// TIA Portal project "Packaging of cubes" (V16)

(* hardware
DEVICE "HMI_1"  TP1200 Comfort
   slot 0: "HMI_1"  TP1200 Comfort  6AV2 124-0MC01-0AX0  16.0.0.0
   slot 1: "HMI_RT_1"  TP1200 Comfort  6AV2 124-0MC01-0AX0  16.0.0.0
   slot 5: "HMI_1.IE_CP_1"  PROFINET Interface  16.0.0.0
      slot 1: "PROFINET Interface_1"  PROFINET Interface
         slot 1: "Port_1"  Port
         slot 2: "Port_2"  Port
   slot 7: "HMI_1.MPI/DP_CP_1"  MPI/DP Interface  16.0.0.0
DEVICE "S71500/ET200MP station_1"  S7-1500 station
   slot 0: "Rail_0"  Rack  6ES7 590-1***0-0AA0
   slot 1: "PLC_1"  CPU 1511-1 PN  6ES7 511-1AK02-0AB0  V2.8
      slot 3: "CPU display_1"  6ES7591-1AA00-0AA0
      slot 32768: "PROFINET interface_1"  X1
         slot 32769: "Port_1"  X1 P1
         slot 32770: "Port_2"  X1 P2
      slot 34817: "Virtual CP interface port_1"  Virtual CP interface port  Virtual CP interface port
*)

// ===== PLC "PLC_1"  CPU 1511-1 PN =====

VAR_GLOBAL   // PLC tag table "Default tag table"
   "Green Cubes Sensor" AT %M0.0 : Bool;
   "Blue Cubes Sensor" AT %M0.1 : Bool;
   "Box not yet Full" AT %M0.2 : Bool;
   "Box Capacity" AT %M2.7 : Bool;
   "Upper Conveyor" AT %M0.4 : Bool;
   "Lower Conveyor" AT %M0.5 : Bool;
   "Box Conveyor" AT %M0.6 : Bool;
   "Box Changing" AT %M0.7 : Bool;
   "Start" AT %M2.0 : Bool;
   "PTRIG1" AT %M2.1 : Bool;
   "Box Sensor" AT %M2.2 : Bool;
   "PTRIG2" AT %M2.3 : Bool;
   "PTRIG3" AT %M2.4 : Bool;
   "PTRIG4" AT %M2.5 : Bool;
   "PTRIG5" AT %M2.6 : Bool;
   "toplam_kutu" AT %MW4 : Int;
   "ToplamMalzeme" AT %MW6 : Int;
   "PTRIG6" AT %M0.3 : Bool;
END_VAR

// folder: System blocks/Program resources

DATA_BLOCK "IEC_Counter_0_DB_2"   // DB1
{ S7_Optimized_Access := 'TRUE' }
AUTHOR : Simatic
FAMILY : IEC
NAME : CNTR
VERSION : 1.0
// stored: InstanceOfName IEC_COUNTER
"IEC_COUNTER"
BEGIN
END_DATA_BLOCK

DATA_BLOCK "IEC_Counter_0_DB"   // DB3
{ S7_Optimized_Access := 'TRUE' }
AUTHOR : Simatic
FAMILY : IEC
NAME : CNTR
VERSION : 1.0
// stored: InstanceOfName IEC_COUNTER
"IEC_COUNTER"
BEGIN
END_DATA_BLOCK

DATA_BLOCK "IEC_Counter_0_DB_1"   // DB4
{ S7_Optimized_Access := 'TRUE' }
AUTHOR : Simatic
FAMILY : IEC
NAME : CNTR
VERSION : 1.0
// stored: InstanceOfName IEC_COUNTER
"IEC_COUNTER"
BEGIN
END_DATA_BLOCK

DATA_BLOCK "IEC_Timer_0_DB_4"   // DB7
{ S7_Optimized_Access := 'TRUE' }
AUTHOR : Simatic
FAMILY : IEC
NAME : IEC_TMR
VERSION : 1.0
// stored: InstanceOfName IEC_TIMER
"IEC_TIMER"
BEGIN
END_DATA_BLOCK

// folder: (top level)

ORGANIZATION_BLOCK "Main"   // OB1, LAD, ProgramCycle
TITLE = "Main Program Sweep (Cycle)"
{ S7_Optimized_Access := 'TRUE' }
VERSION : 0.1
   VAR_INPUT
      Initial_Call : Bool;   // Initial call of this OB
      Remanence : Bool;   // =True, if remanent data are available
   END_VAR
   VAR_TEMP
      BoxCapacity1 : Bool;
   END_VAR
   VAR_TEMP   // added for the SCL form of the ladder/FBD networks
      _w1 : Bool;
      _w2 : Bool;
   END_VAR
BEGIN

REGION Network 1
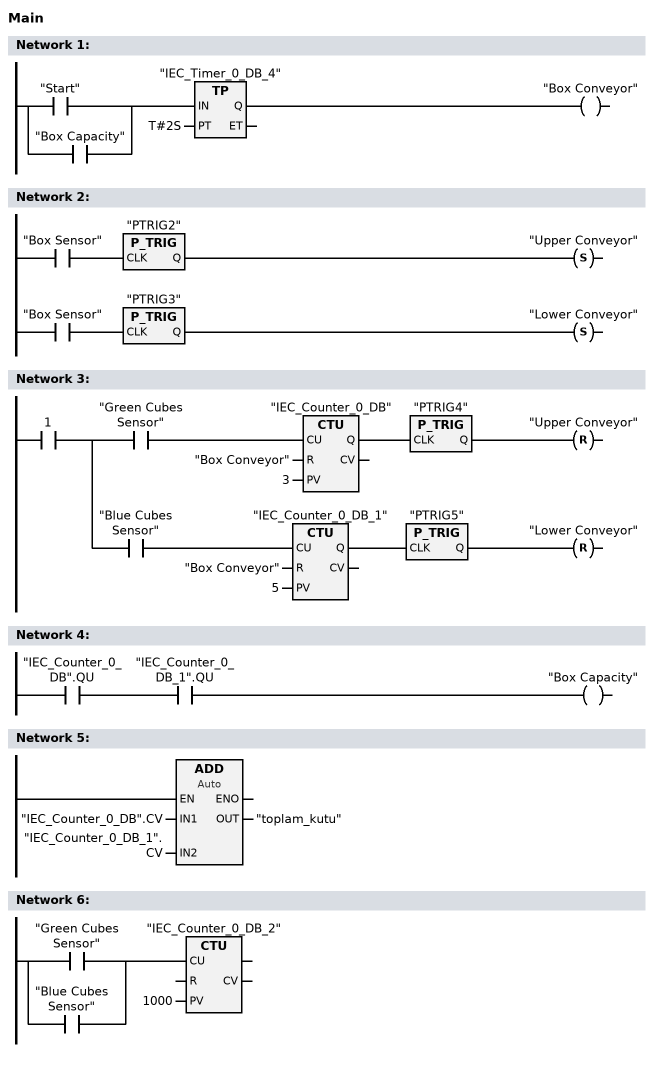
   "IEC_Timer_0_DB_4".TP(IN := "Start" OR "Box Capacity", PT := T#2S);
   "Box Conveyor" := "IEC_Timer_0_DB_4".Q;
END_REGION

REGION Network 2
   RUNG wire#powerrail
      Contact( "Box Sensor" )
      P_Trig( "PTRIG2" )
      S_Coil( "Upper Conveyor" )
   END_RUNG
   RUNG wire#powerrail
      Contact( "Box Sensor" )
      P_Trig( "PTRIG3" )
      S_Coil( "Lower Conveyor" )
   END_RUNG
   // the same network as SCL:
   #_w1 := "Box Sensor" AND NOT "PTRIG2";   // rising edge
   "PTRIG2" := "Box Sensor";
   IF #_w1 THEN "Upper Conveyor" := TRUE; END_IF;
   #_w2 := "Box Sensor" AND NOT "PTRIG3";   // rising edge
   "PTRIG3" := "Box Sensor";
   IF #_w2 THEN "Lower Conveyor" := TRUE; END_IF;
END_REGION

REGION Network 3
   "IEC_Counter_0_DB".CTU(CU := 1 AND "Green Cubes Sensor", R := "Box Conveyor", PV := 3);
   #_w1 := "IEC_Counter_0_DB".Q AND NOT "PTRIG4";   // rising edge
   "PTRIG4" := "IEC_Counter_0_DB".Q;
   IF #_w1 THEN "Upper Conveyor" := FALSE; END_IF;
   "IEC_Counter_0_DB_1".CTU(CU := 1 AND "Blue Cubes Sensor", R := "Box Conveyor", PV := 5);
   #_w2 := "IEC_Counter_0_DB_1".Q AND NOT "PTRIG5";   // rising edge
   "PTRIG5" := "IEC_Counter_0_DB_1".Q;
   IF #_w2 THEN "Lower Conveyor" := FALSE; END_IF;
END_REGION

REGION Network 4
   RUNG wire#powerrail
      Contact( "IEC_Counter_0_DB".QU )
      Contact( "IEC_Counter_0_DB_1".QU )
      Coil( "Box Capacity" )
   END_RUNG
   // the same network as SCL:
   "Box Capacity" := "IEC_Counter_0_DB".QU AND "IEC_Counter_0_DB_1".QU;
END_REGION

REGION Network 5
   RUNG wire#powerrail
      Add(in1 := "IEC_Counter_0_DB".CV, in2 := "IEC_Counter_0_DB_1".CV, out => "toplam_kutu")
   END_RUNG
   // the same network as SCL:
   "toplam_kutu" := "IEC_Counter_0_DB".CV + "IEC_Counter_0_DB_1".CV;
END_REGION

REGION Network 6
   "IEC_Counter_0_DB_2".CTU(CU := "Green Cubes Sensor" OR "Blue Cubes Sensor", PV := 1000);
END_REGION
END_ORGANIZATION_BLOCK

(* ===== HMI "HMI_RT_1" =====
system functions are stored by id; their names below are inferred from use
connection "HMI_Connection_1": ETHERNET, S7_1500_OMS

HMI tags "Default tag table"
   "Tag_ScreenNumber" : UInt, internal
   "Start" : Bool = PLC Start AT %M2.0, 1 s
   "Upper Conveyor" : Bool = PLC "Upper Conveyor" AT %M0.4, 1 s
   "Lower Conveyor" : Bool = PLC "Lower Conveyor" AT %M0.5, 1 s
   "Box Capacity" : Bool = PLC "Box Capacity" AT %M2.7, 1 s
   "Green Cubes Sensor" : Bool = PLC "Green Cubes Sensor" AT %M0.0, 1 s
   "Blue Cubes Sensor" : Bool = PLC "Blue Cubes Sensor" AT %M0.1, 1 s
   "Box Conveyor" : Bool = PLC "Box Conveyor" AT %M0.6, 1 s
   "Box Sensor" : Bool = PLC "Box Sensor" AT %M2.2, 1 s
   "IEC_Counter_0_DB_CV" : Int = PLC IEC_Counter_0_DB.CV, 1 s
   "IEC_Counter_0_DB_1_CV" : Int = PLC IEC_Counter_0_DB_1.CV, 1 s
   "toplam_kutu" : Int = PLC toplam_kutu AT %MW4, 1 s
   "ToplamMalzeme" : Int = PLC ToplamMalzeme AT %MW6, 1 s
   "IEC_Counter_0_DB_2_CV" : Int = PLC IEC_Counter_0_DB_2.CV, 1 s

screen "Root screen" 1280x740, template "Template_1"
   on GenerateScreen: InvertBit("Start")
   TextField "Text field_1" at 7,37 size 182x37; Text 'Upper Conveyor :'
   TextField "Text field_2" at 6,153 size 183x37; Text 'Lower Conveyor :'
   Circle "Circle_1" at 228,29 size 48x48
      Appearance <- "Upper Conveyor"
   Circle "Circle_2" at 228,142 size 48x48
      Appearance <- "Lower Conveyor"
   TextField "Text field_3" at 8,241 size 153x37; Text 'Box Capacity :'
   IOField "I/O field_1" at 213,241 size 96x32; FormatPattern s99999
      ProcessValue <- "toplam_kutu"
   TextField "Text field_4" at 6,316 size 208x35; Text 'Green Cube Sensor :'
   TextField "Text field_5" at 6,378 size 200x35; Text 'Blue Cube Sensor :'
   GraphicView "Graphic view_3" at 333,113 size 91x92; Picture "Graphic_3"
   GraphicView "Graphic view_1" at 326,7 size 96x92; Picture "Graphic_4"
   IOField "I/O field_2" at 224,316 size 96x32; FormatPattern s99999
      ProcessValue <- "IEC_Counter_0_DB_CV"
   IOField "I/O field_3" at 224,378 size 96x32; FormatPattern s99999
      ProcessValue <- "IEC_Counter_0_DB_1_CV"
   Button "Button_3" at 506,39 size 206x32; TextOff 'Start'
      on Press: function_b14e0dd5("Start", 0)
   Circle "Circle_3" at 755,26 size 48x48
      Appearance <- "Start"
   TextField "Text field_6" at 8,455 size 159x35; Text 'Box Conveyor :'
   Circle "Circle_4" at 236,446 size 48x48
      Appearance <- "Box Conveyor"
   TextField "Text field_7" at 7,523 size 135x35; Text 'Box Sensor :'
   Circle "Circle_5" at 345,365 size 48x48
      Appearance <- "Blue Cubes Sensor"
   Button "Button_1" at 194,523 size 96x32; TextOff 'Box sensör'
      on Press: function_b14e0dd5("Box Sensor", 0)
   Button "Button_2" at 417,316 size 96x32; TextOff 'Text'
      on Press: function_b14e0dd5("Green Cubes Sensor", 0)
   Button "Button_4" at 417,378 size 96x32; TextOff 'Text'
      on Press: function_b14e0dd5("Blue Cubes Sensor", 0)
   TextField "Text field_8" at 11,598 size 175x25; Text 'Toplam Malzeme :'
   IOField "I/O field_4" at 194,594 size 96x32; FormatPattern s99999
      ProcessValue <- "IEC_Counter_0_DB_2_CV"

Template "Template_1" 1280x740
   Button "Exit" at 1200,679 size 78x59; TextOff 'Exit'; PictureOff "ExitRuntime_TP1200_Comfort_TR"; PictureOn "ExitRuntime_TP1200_Comfort_TR"
      on Release: StopRuntime(0)
   Button "Template_Button" at 1120,679 size 78x59; TextOff 'Text'
   Button "Template_Button_1" at 1040,679 size 78x59; TextOff 'Text'
   Button "Template_Button_2" at 960,679 size 78x59; TextOff 'Text'
   Button "Template_Button_3" at 880,679 size 78x59; TextOff 'Text'
   Button "Template_Button_4" at 800,679 size 78x59; TextOff 'Text'
   Button "Template_Button_5" at 720,679 size 78x59; TextOff 'Text'
   Button "Template_Button_6" at 640,679 size 78x59; TextOff 'Text'
   Button "Template_Button_7" at 561,679 size 78x59; TextOff 'Text'
   Button "Template_Button_8" at 481,679 size 78x59; TextOff 'Text'
   Button "Template_Button_9" at 401,679 size 78x59; TextOff 'Text'
   Button "Template_Button_10" at 321,679 size 78x59; TextOff 'Text'
   Button "Template_Button_11" at 241,679 size 78x59; TextOff 'Text'
   Button "Template_Button_12" at 161,679 size 78x59; TextOff 'Text'
   Button "Template_Button_13" at 81,679 size 78x59; TextOff 'Text'
   Button "Start screen" at 1,679 size 78x59; TextOff 'Start screen'; PictureOff "NavigateHome_TP1200_Comfort_TR"; PictureOn "NavigateHome_TP1200_Comfort_TR"
      on Release: ActivateScreen("Root screen", 0)
*)